// TwinCAT 3 PLC project PLC
// ProgramVersion: 3.1.4026.22
// libraries:
//   Tc2_Standard, * (Beckhoff Automation GmbH)
//   Tc2_System, * (Beckhoff Automation GmbH)
//   Tc2_Utilities, * (Beckhoff Automation GmbH)
//   Tc3_EventLogger, * (Beckhoff Automation GmbH)
// project tree:
//   / PlcTask.TcTTO
//   POUs/ MAIN.TcPOU
// real-time tasks:
//   TASK PlcTask: cycle T#10ms, priority 20, ADS port 350
// I/O:
//   DEVICE Device 1 (EtherCAT), AmsNetId 192.168.2.60.2.1
//     Term 1 (EK1100) [EK1100 EtherCAT Coupler (2A E-Bus)]
//       Term 2 (EL1859) [EL1859 8Ch. Dig. Input 24V, 3ms, 8Ch. Dig. Output 24V, 0.5A]
//       Term 3 (EL3255) [EL3255 5Ch. potentiometer measurement with sensor supply]
//       Term 4 (EL4374) [EL4374 2Ch. Ana. Input, 2Ch. Ana. Output, +/-10V, +/-20mA, 16 Bit]
//       Term 5 (EL9011) [EL9011 End Terminal]
// variable links:
//   PLC/PLC Instance <-> Device 1 (EtherCAT)/Term 1 (EK1100)/Term 3 (EL3255)
//     PlcTask Inputs/MAIN.iPotentiometerValue <-> AI Standard Channel 1/Value

CONFIGURATION PLC
    RESOURCE PLC ON TwinCAT3
        TASK PlcTask(INTERVAL := T#10ms, PRIORITY := 20);
        PROGRAM MAIN WITH PlcTask : MAIN;
    END_RESOURCE
END_CONFIGURATION

// ---- POUs/MAIN.TcPOU
PROGRAM MAIN
VAR

	// Flag para el control del primer ciclo de escaneo (inicialización)
	xInit					:BOOL:=TRUE;
	
	// Instancias para la gestión de alarmas y mensajes del sistema
	fbAlarm					:FB_TcAlarm;
	fbMsg					:FB_TcMessage;	
	fbPotentiometerMsg		:FB_TcMessage; // Mensaje específico para el registro del potenciómetro

	// Variables para la generación automática de eventos de prueba
	xCreateLogEntries		:BOOL;               			
	tonPulse				:TON;           	    	
	iCnt					:INT;
	
	// Variables asociadas al hardware y lectura del potenciómetro
	fbDeviceInfo			:FB_GetDeviceIdentificationEx;
	xTriggerInput			:BOOL;         // Entrada física digital para el disparo del registro
	rtTrigger				:R_TRIG;       // Detector de flanco de subida para la entrada digital
	iPotentiometerValue		AT %I* :INT;          // Valor analógico actual del potenciómetro
	
	// Variables de configuración de rutas y archivos de exportación
	sExportPath				:STRING(255);
	sFullPathName			:STRING(255);
	xExportLog				:BOOL;
	
	// Tipos enumerados para el control de la secuencia y filtrado
	FilterExample			:(NONE,OnlyMsg,OnlyAlarm,Complex):=OnlyAlarm;	                    	
	ExportStep				:(IDEL,SetFilters,Export);
	
	// Componentes globales del TwinCAT Event Logger
	fbTcEventLogger			:FB_TcEventLogger;
	fbCsvExportSetting		:FB_TcEventCsvExportSettings;
	fbExportFilter			:FB_TcEventFilter;
	hrDebug					:HRESULT;
	
	// Variables para la gestión y formateo de la marca de tiempo
	TimeSource				:(SystemTime,LocalSystemTime);
	fbGetTime				:FB_LocalSystemTime;
	dtNow					:DT;
	sNow					:STRING;
	dtFilterTimeGT			:DT;

	// Diagnóstico del proceso de exportación
	xExportError			:BOOL;
	hrExportErrorCode		:HRESULT;
	iExportBusyCnt			:UDINT;
	
	// Variables para el vaciado de registros del sistema
	xClearLoggedEvents		:BOOL;
	xClearLoggedEventsError :BOOL;
	hrClearLoggedEventsErrorCode :HRESULT;
	iBusyClearing			:BOOL;
END_VAR
VAR CONSTANT
	// Constantes de caracteres utilizadas para el formateo de cadenas de texto
	sDT						:STRING(3):='DT#';
	sColon					:STRING(1):=':';
	sUnderScope				:STRING(1):='_';
END_VAR

// Inicialización de componentes
IF xInit THEN
	xInit:=FALSE;
	
	fbAlarm.CreateEx(TC_EVENTS.MyEvents.Alarm,FALSE,0);
	fbMsg.CreateEx(TC_EVENTS.MyEvents.Msg,0);
	fbPotentiometerMsg.CreateEx(TC_EVENTS.MyEvents.PotentiometerLog,0);
	
	fbDeviceInfo(bExecute:=TRUE);
END_IF

fbDeviceInfo();

IF NOT fbDeviceInfo.bError THEN
	fbDeviceInfo.bExecute:=FALSE;
END_IF


// Registro de potenciómetro por entrada digital
rtTrigger(CLK := xTriggerInput);

IF rtTrigger.Q THEN
	fbPotentiometerMsg.ipArguments.Clear().AddInt(iPotentiometerValue);
	fbPotentiometerMsg.Send(0);
	xTriggerInput := False;
END_IF


// Generación de eventos de prueba
tonPulse(IN:=NOT tonPulse.Q AND xCreateLogEntries, PT:=T#200MS);

IF tonPulse.Q THEN
	iCnt:=iCnt+1;
	
	IF fbAlarm.bRaised THEN
		fbAlarm.Clear(0,TRUE);
	END_IF
	
	fbAlarm.ipArguments.Clear().AddInt(iCnt);
	fbAlarm.Raise(0);
	
	fbMsg.ipArguments.Clear().AddInt(iCnt);
	fbMsg.Send(0);
END_IF

IF iCnt>=10 THEN
	xCreateLogEntries	:=FALSE;
	iCnt				:=0;
END_IF


// Gestión de tiempo del sistema y formato de cadena
dtNow	:= FILETIME64_TO_DT(F_GetSystemTime());	
sNow	:= DT_TO_STRING(dtNow);

FindAndDelete(pSrcString:= ADR(sNow),ADR(sDT),ADR(sNow),SIZEOF(sNow));
FindAndReplace(pSrcString:= ADR(sNow),pDeleteString:=ADR(sColon),pInsertString:=ADR(sUnderScope),pDstString:=ADR(sNow),nDstSize:=SIZEOF(sNow));
	

// Máquina de estados: Exportación a CSV
CASE ExportStep OF
	
	IDEL:
		IF xExportLog THEN
			xExportLog 		:=FALSE;	
			ExportStep		:=SetFilters;		
		END_IF	
	
	SetFilters:	
		// Definición de la ruta según el sistema operativo detectado
		IF fbDeviceInfo.stDevIdent.strImageOsName = 'Windows CE' THEN
			sExportPath:='\Hard Disk\TwinCAT\3.1\Boot\';
		ELSIF FIND(fbDeviceInfo.stDevIdent.strImageOsName,'Windows 10')>0 THEN
			sExportPath:='C:\Users\Administrator\Documents\CSV\';
		ELSIF fbDeviceInfo.stDevIdent.strImageOsName='TC/BSD' THEN
			sExportPath:='/usr/local/etc/TwinCAT/3.1/Boot/';
		END_IF
		
		sFullPathName	:=CONCAT(sExportPath,CONCAT(CONCAT('LogExport',sNow),'.csv'));		

		fbCsvExportSetting.Clear();
		fbCsvExportSetting.sDelimiter:=',';
		
		fbCsvExportSetting.AddField(eType:=TcEventField.EventText, 'Event Text', '', );
		
		fbCsvExportSetting.AddField(eType:=TcEventField.TimeRaised, 'Time Raised', '', );
		fbCsvExportSetting.AddField(eType:=TcEventField.TimeConfirmed, 'Time Confirmed', '', );
		fbCsvExportSetting.AddField(eType:=TcEventField.TimeCleared, 'Time Cleared', '', );
		fbCsvExportSetting.AddField(eType:=TcEventField.SeverityLevel, 'Severity', '', );	
		fbCsvExportSetting.AddField(eType:=TcEventField.SourceName, 'Source', '', );		
		fbCsvExportSetting.AddFilter(fbExportFilter); 
		
		FilterExample := OnlyMsg;
	
		CASE FilterExample OF
			NONE:
				fbExportFilter.Clear();
			OnlyMsg:
				fbExportFilter.Clear().IsMessage();
			OnlyAlarm:
				fbExportFilter.Clear().IsAlarm();		
			Complex:
				fbExportFilter.Clear().IsAlarm().AND_OP().TimeRaised.GreaterThan(DT_TO_FILETIME64(dtFilterTimeGT));
		END_CASE

		iExportBusyCnt	:=0;
		ExportStep		:=Export;
		
	Export:
		// Ejecución de la exportación asíncrona
		IF fbTcEventLogger.ExportLoggedEvents(	sFileName		 :=sFullPathName ,
		 										ipExportSettings :=fbCsvExportSetting , 
												bError			 =>xExportError , 
												hrErrorCode		 =>hrExportErrorCode ) 
		THEN
			ExportStep:=IDEL;
		ELSE
			iExportBusyCnt:=iExportBusyCnt+1;
		END_IF
		
END_CASE


// Vaciado de registros de eventos
IF xClearLoggedEvents THEN
	fbTcEventLogger.ClearAllAlarms(0,TRUE);
	
	IF fbTcEventLogger.ClearLoggedEvents(ipClearSettings:=0 , bError=>xClearLoggedEventsError , hrErrorCode=>hrClearLoggedEventsErrorCode )THEN
		xClearLoggedEvents	:=FALSE;
		iBusyClearing		:=FALSE;
	ELSE
		iBusyClearing		:=TRUE;
	END_IF
END_IF

END_PROGRAM
